FUNCTION_BLOCK FB_ValveControl
VAR_INPUT
END_VAR
VAR_OUTPUT
END_VAR
VAR
END_VAR

END_FUNCTION_BLOCK

(* stored: Version 1.1.0.1, ProductVersion 3.1.4024.12
   POU FB_ValveControl: Id {13a96f09-3b20-4f3b-b174-6aae60c0a541}, SpecialFunc None *)
